{attribute 'qualified_only'}
{attribute 'strict'}
TYPE eAcInputType :
(
	None 	:= 0,
	Grid 	:= 1,
	Genset	:= 2
);
END_TYPE

(* stored: Version 1.1.0.1, ProductVersion 3.1.4026.18
   DUT eAcInputType: Id {d04b834f-1968-47c1-971a-bb64973b36b8} *)
